TYPE T_PROCESS : DWORD; END_TYPE

(* stored: Version 1.1.0.1, ProductVersion 3.1.4026.18
   DUT T_PROCESS: Id {13d73441-74ca-4c91-9744-668e0f7fb106} *)
